// TIA Portal V19 export
DATA_BLOCK "WeldReg_PERS"   // DB168
// stored: MemoryReserve 100
   VAR RETAIN
      PersistentValues : "udt_WeldReg_Pers";
   END_VAR
BEGIN
END_DATA_BLOCK
